// TIA Portal V19 export
FUNCTION_BLOCK "Area01_HU_FB"   // FB38, LAD
TITLE = AREA 01 HU PUMP
// stored: MemoryReserve 100, SetENOAutomatically false
   VAR_INPUT
      AreaInterface : "AreaInterface";
   END_VAR
   VAR_OUTPUT
      MachineInterface : "MachineInterface";
   END_VAR
   VAR
      Pump : "HU_Pump";
      Tank { S7_SetPoint := 'True'} : "HU_Tank";
      HMI : Struct
         Pressure_CoilCar : Real;
         Pressure_Peeler : Real;
         Pressure_JB_Cut : Real;
      END_STRUCT;
   END_VAR
   VAR_TEMP
      retval : Int;
      OilTemperature : Real;
      AnalTemperature_Real : Real;
      Delta : Real;
      Delta2 : Real;
   END_VAR
BEGIN

REGION Network 1: <<< PUMP >>>
END_REGION

REGION Network 2: Data In
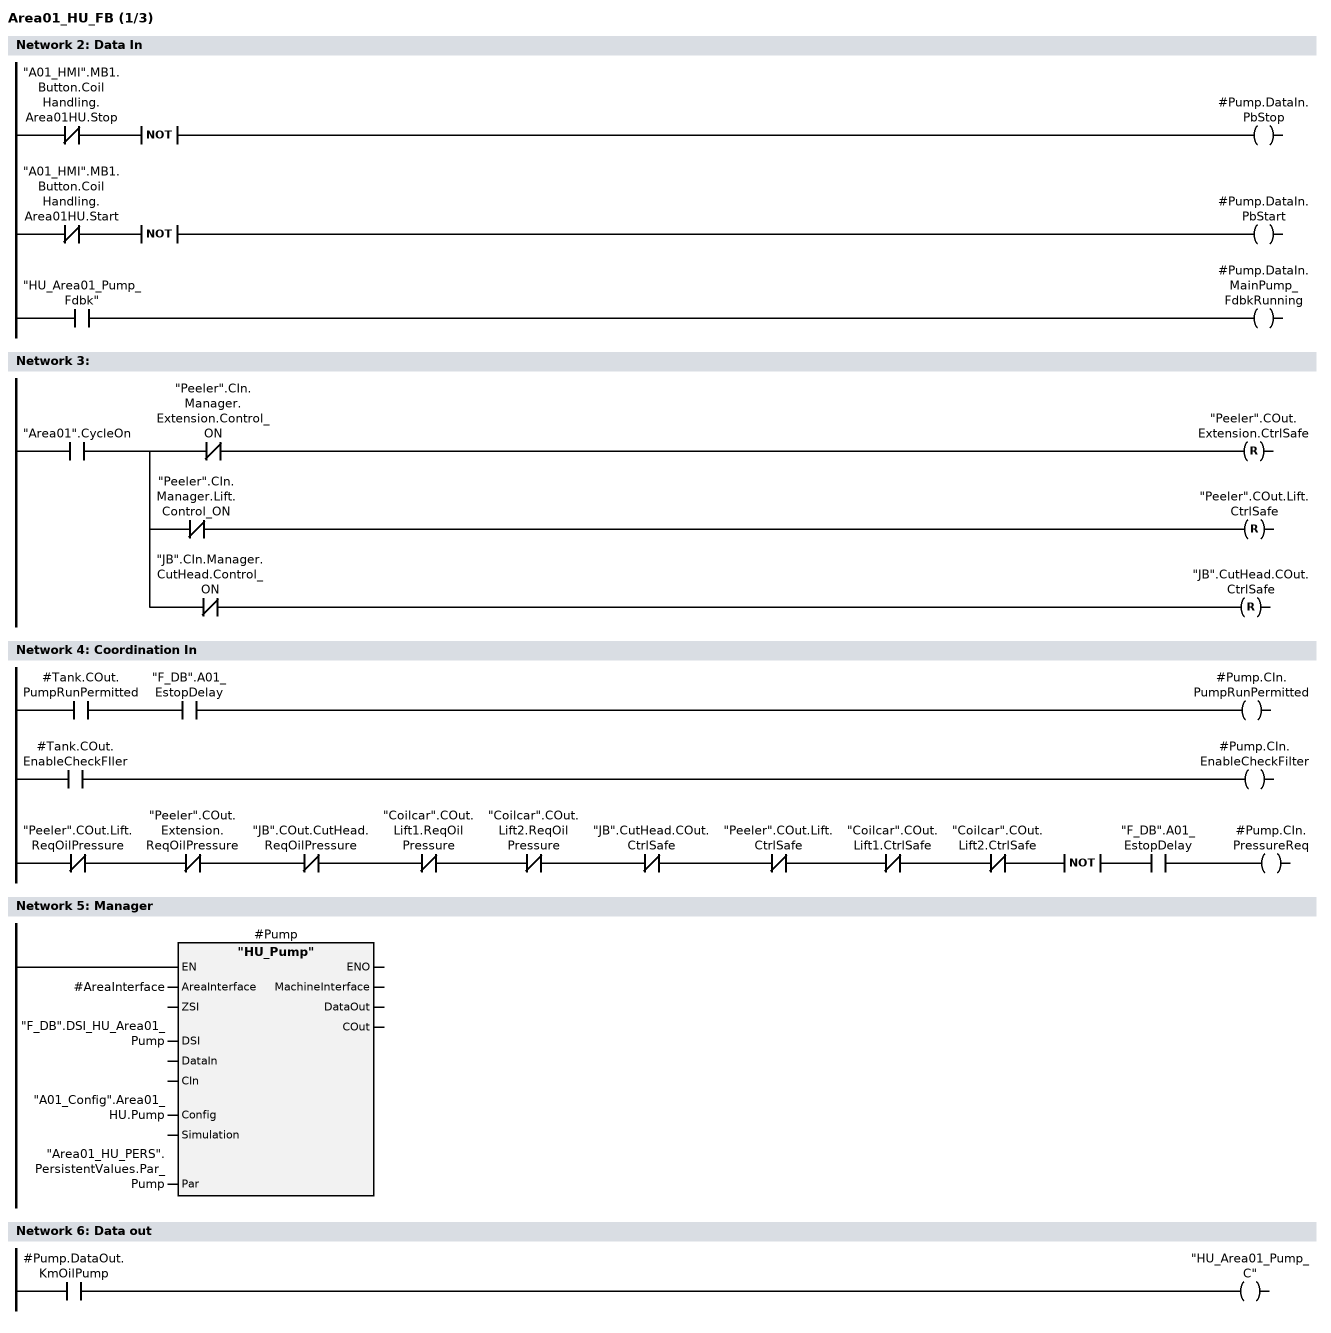
   RUNG wire#powerrail
      I_Contact( "A01_HMI".MB1.Button.CoilHandling.Area01HU.Stop )
      Not()
      Coil( #Pump.DataIn.PbStop )
   END_RUNG
   RUNG wire#powerrail
      I_Contact( "A01_HMI".MB1.Button.CoilHandling.Area01HU.Start )
      Not()
      Coil( #Pump.DataIn.PbStart )
   END_RUNG
   RUNG wire#powerrail
      Contact( "HU_Area01_Pump_Fdbk" )
      Coil( #Pump.DataIn.MainPump_FdbkRunning )
   END_RUNG
   // the same network as SCL:
   #Pump.DataIn.PbStop := NOT (NOT "A01_HMI".MB1.Button.CoilHandling.Area01HU.Stop);
   #Pump.DataIn.PbStart := NOT (NOT "A01_HMI".MB1.Button.CoilHandling.Area01HU.Start);
   #Pump.DataIn.MainPump_FdbkRunning := "HU_Area01_Pump_Fdbk";
END_REGION

REGION Network 3
   RUNG wire#powerrail
      Contact( "Area01".CycleOn )
      wire#w1
      I_Contact( "Peeler".CIn.Manager.Extension.Control_ON )
      R_Coil( "Peeler".COut.Extension.CtrlSafe )
   END_RUNG
   RUNG wire#w1
      I_Contact( "Peeler".CIn.Manager.Lift.Control_ON )
      R_Coil( "Peeler".COut.Lift.CtrlSafe )
   END_RUNG
   RUNG wire#w1
      I_Contact( "JB".CIn.Manager.CutHead.Control_ON )
      R_Coil( "JB".CutHead.COut.CtrlSafe )
   END_RUNG
   // the same network as SCL:
   IF "Area01".CycleOn AND NOT "Peeler".CIn.Manager.Extension.Control_ON THEN
       "Peeler".COut.Extension.CtrlSafe := FALSE;
   END_IF;
   IF "Area01".CycleOn AND NOT "Peeler".CIn.Manager.Lift.Control_ON THEN
       "Peeler".COut.Lift.CtrlSafe := FALSE;
   END_IF;
   IF "Area01".CycleOn AND NOT "JB".CIn.Manager.CutHead.Control_ON THEN
       "JB".CutHead.COut.CtrlSafe := FALSE;
   END_IF;
END_REGION

REGION Network 4: Coordination In
   RUNG wire#powerrail
      Contact( #Tank.COut.PumpRunPermitted )
      Contact( "F_DB".A01_EstopDelay )
      Coil( #Pump.CIn.PumpRunPermitted )
   END_RUNG
   RUNG wire#powerrail
      Contact( #Tank.COut.EnableCheckFIler )
      Coil( #Pump.CIn.EnableCheckFilter )
   END_RUNG
   RUNG wire#powerrail
      I_Contact( "Peeler".COut.Lift.ReqOilPressure )
      I_Contact( "Peeler".COut.Extension.ReqOilPressure )
      I_Contact( "JB".COut.CutHead.ReqOilPressure )
      I_Contact( "Coilcar".COut.Lift1.ReqOilPressure )
      I_Contact( "Coilcar".COut.Lift2.ReqOilPressure )
      I_Contact( "JB".CutHead.COut.CtrlSafe )
      I_Contact( "Peeler".COut.Lift.CtrlSafe )
      I_Contact( "Coilcar".COut.Lift1.CtrlSafe )
      I_Contact( "Coilcar".COut.Lift2.CtrlSafe )
      Not()
      Contact( "F_DB".A01_EstopDelay )
      Coil( #Pump.CIn.PressureReq )
   END_RUNG
   // the same network as SCL:
   #Pump.CIn.PumpRunPermitted := #Tank.COut.PumpRunPermitted AND "F_DB".A01_EstopDelay;
   #Pump.CIn.EnableCheckFilter := #Tank.COut.EnableCheckFIler;
   #Pump.CIn.PressureReq := NOT (NOT "Peeler".COut.Lift.ReqOilPressure AND NOT "Peeler".COut.Extension.ReqOilPressure AND NOT "JB".COut.CutHead.ReqOilPressure AND NOT "Coilcar".COut.Lift1.ReqOilPressure AND NOT "Coilcar".COut.Lift2.ReqOilPressure AND NOT "JB".CutHead.COut.CtrlSafe AND NOT "Peeler".COut.Lift.CtrlSafe AND NOT "Coilcar".COut.Lift1.CtrlSafe AND NOT "Coilcar".COut.Lift2.CtrlSafe) AND "F_DB".A01_EstopDelay;
END_REGION

REGION Network 5: Manager
   RUNG wire#powerrail
      #Pump(AreaInterface := #AreaInterface, ZSI :=, DSI := "F_DB".DSI_HU_Area01_Pump, DataIn :=, CIn :=, Config := "A01_Config".Area01_HU.Pump, Simulation :=, Par := "Area01_HU_PERS".PersistentValues.Par_Pump, MachineInterface =>, DataOut =>, COut =>)
   END_RUNG
   // the same network as SCL:
   #Pump(AreaInterface := #AreaInterface,   // "HU_Pump"
         DSI := "F_DB".DSI_HU_Area01_Pump,
         Config := "A01_Config".Area01_HU.Pump,
         Par := "Area01_HU_PERS".PersistentValues.Par_Pump);
END_REGION

REGION Network 6: Data out
   RUNG wire#powerrail
      Contact( #Pump.DataOut.KmOilPump )
      Coil( "HU_Area01_Pump_C" )
   END_RUNG
   // the same network as SCL:
   "HU_Area01_Pump_C" := #Pump.DataOut.KmOilPump;
END_REGION

REGION Network 7: >
END_REGION

REGION Network 8: >
END_REGION

REGION Network 9: >
END_REGION

REGION Network 10: <<< TANK >>>
END_REGION

REGION Network 11: Data In
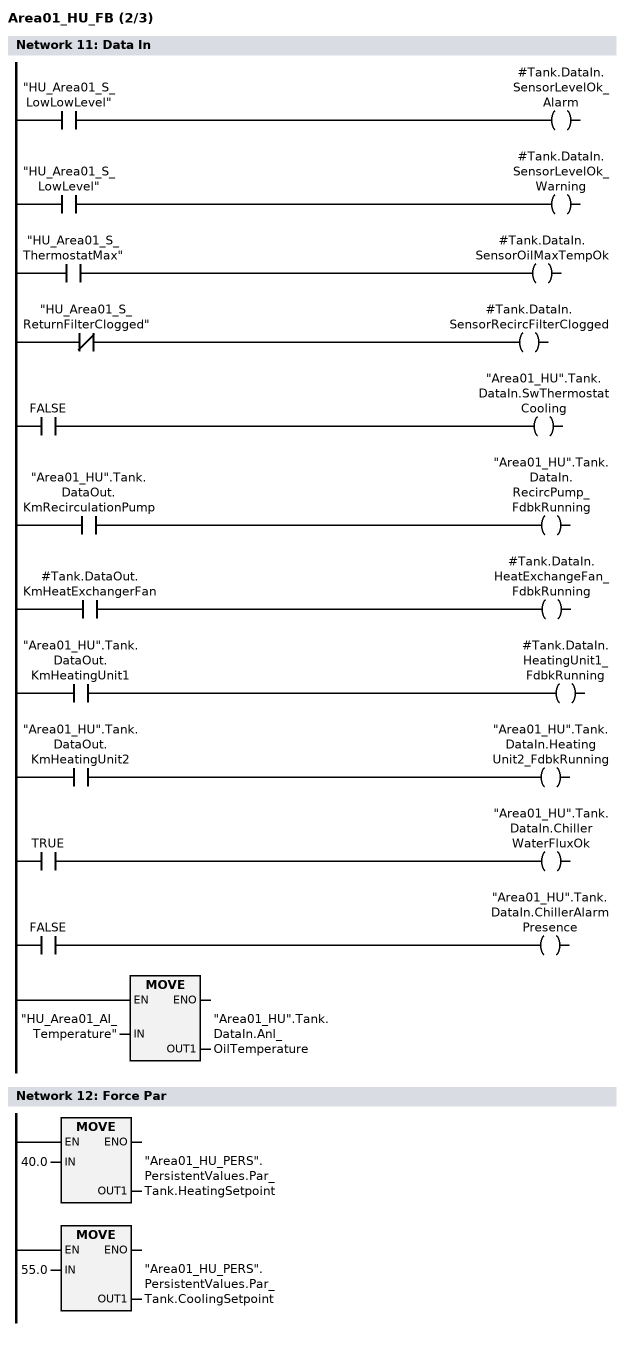
   RUNG wire#powerrail
      Contact( "HU_Area01_S_LowLowLevel" )
      Coil( #Tank.DataIn.SensorLevelOk_Alarm )
   END_RUNG
   RUNG wire#powerrail
      Contact( "HU_Area01_S_LowLevel" )
      Coil( #Tank.DataIn.SensorLevelOk_Warning )
   END_RUNG
   RUNG wire#powerrail
      Contact( "HU_Area01_S_ThermostatMax" )
      Coil( #Tank.DataIn.SensorOilMaxTempOk )
   END_RUNG
   RUNG wire#powerrail
      I_Contact( "HU_Area01_S_ReturnFilterClogged" )
      Coil( #Tank.DataIn.SensorRecircFilterClogged )
   END_RUNG
   RUNG wire#powerrail
      Contact( FALSE )
      Coil( "Area01_HU".Tank.DataIn.SwThermostatCooling )
   END_RUNG
   RUNG wire#powerrail
      Contact( "Area01_HU".Tank.DataOut.KmRecirculationPump )
      Coil( "Area01_HU".Tank.DataIn.RecircPump_FdbkRunning )
   END_RUNG
   RUNG wire#powerrail
      Contact( #Tank.DataOut.KmHeatExchangerFan )
      Coil( #Tank.DataIn.HeatExchangeFan_FdbkRunning )
   END_RUNG
   RUNG wire#powerrail
      Contact( "Area01_HU".Tank.DataOut.KmHeatingUnit1 )
      Coil( #Tank.DataIn.HeatingUnit1_FdbkRunning )
   END_RUNG
   RUNG wire#powerrail
      Contact( "Area01_HU".Tank.DataOut.KmHeatingUnit2 )
      Coil( "Area01_HU".Tank.DataIn.HeatingUnit2_FdbkRunning )
   END_RUNG
   RUNG wire#powerrail
      Contact( TRUE )
      Coil( "Area01_HU".Tank.DataIn.ChillerWaterFluxOk )
   END_RUNG
   RUNG wire#powerrail
      Contact( FALSE )
      Coil( "Area01_HU".Tank.DataIn.ChillerAlarmPresence )
   END_RUNG
   RUNG wire#powerrail
      Move(in := "HU_Area01_AI_Temperature", out1 => "Area01_HU".Tank.DataIn.Anl_OilTemperature)
   END_RUNG
   // the same network as SCL:
   #Tank.DataIn.SensorLevelOk_Alarm := "HU_Area01_S_LowLowLevel";
   #Tank.DataIn.SensorLevelOk_Warning := "HU_Area01_S_LowLevel";
   #Tank.DataIn.SensorOilMaxTempOk := "HU_Area01_S_ThermostatMax";
   #Tank.DataIn.SensorRecircFilterClogged := NOT "HU_Area01_S_ReturnFilterClogged";
   "Area01_HU".Tank.DataIn.SwThermostatCooling := FALSE;
   "Area01_HU".Tank.DataIn.RecircPump_FdbkRunning := "Area01_HU".Tank.DataOut.KmRecirculationPump;
   #Tank.DataIn.HeatExchangeFan_FdbkRunning := #Tank.DataOut.KmHeatExchangerFan;
   #Tank.DataIn.HeatingUnit1_FdbkRunning := "Area01_HU".Tank.DataOut.KmHeatingUnit1;
   "Area01_HU".Tank.DataIn.HeatingUnit2_FdbkRunning := "Area01_HU".Tank.DataOut.KmHeatingUnit2;
   "Area01_HU".Tank.DataIn.ChillerWaterFluxOk := TRUE;
   "Area01_HU".Tank.DataIn.ChillerAlarmPresence := FALSE;
   "Area01_HU".Tank.DataIn.Anl_OilTemperature := "HU_Area01_AI_Temperature";
END_REGION

REGION Network 12: Force Par
   RUNG wire#powerrail
      { S7_GenerateENO := "TRUE" } Move(in := 40.0, out1 => "Area01_HU_PERS".PersistentValues.Par_Tank.HeatingSetpoint)
   END_RUNG
   RUNG wire#powerrail
      { S7_GenerateENO := "TRUE" } Move(in := 55.0, out1 => "Area01_HU_PERS".PersistentValues.Par_Tank.CoolingSetpoint)
   END_RUNG
   // the same network as SCL:
   "Area01_HU_PERS".PersistentValues.Par_Tank.HeatingSetpoint := 40.0;
   "Area01_HU_PERS".PersistentValues.Par_Tank.CoolingSetpoint := 55.0;
END_REGION

REGION Network 13: HMI pressure
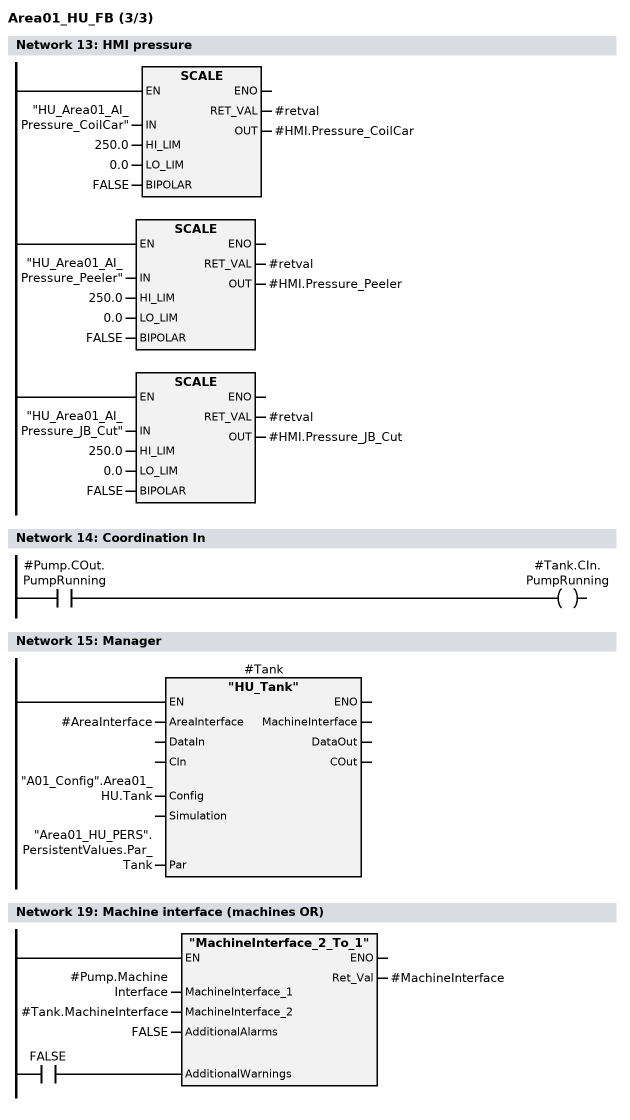
   #retval := SCALE(IN := "HU_Area01_AI_Pressure_CoilCar",
                    HI_LIM := 250.0,
                    LO_LIM := 0.0,
                    BIPOLAR := FALSE,
                    OUT => #HMI.Pressure_CoilCar);
   #retval := SCALE(IN := "HU_Area01_AI_Pressure_Peeler",
                    HI_LIM := 250.0,
                    LO_LIM := 0.0,
                    BIPOLAR := FALSE,
                    OUT => #HMI.Pressure_Peeler);
   #retval := SCALE(IN := "HU_Area01_AI_Pressure_JB_Cut",
                    HI_LIM := 250.0,
                    LO_LIM := 0.0,
                    BIPOLAR := FALSE,
                    OUT => #HMI.Pressure_JB_Cut);
END_REGION

REGION Network 14: Coordination In
   RUNG wire#powerrail
      Contact( #Pump.COut.PumpRunning )
      Coil( #Tank.CIn.PumpRunning )
   END_RUNG
   // the same network as SCL:
   #Tank.CIn.PumpRunning := #Pump.COut.PumpRunning;
END_REGION

REGION Network 15: Manager
   RUNG wire#powerrail
      #Tank(AreaInterface := #AreaInterface, DataIn :=, CIn :=, Config := "A01_Config".Area01_HU.Tank, Simulation :=, Par := "Area01_HU_PERS".PersistentValues.Par_Tank, MachineInterface =>, DataOut =>, COut =>)
   END_RUNG
   // the same network as SCL:
   #Tank(AreaInterface := #AreaInterface,   // "HU_Tank"
         Config := "A01_Config".Area01_HU.Tank,
         Par := "Area01_HU_PERS".PersistentValues.Par_Tank);
END_REGION

REGION Network 16: >
END_REGION

REGION Network 17: >
END_REGION

REGION Network 18: >
END_REGION

REGION Network 19: Machine interface (machines OR)
   RUNG wire#powerrail
      "MachineInterface_2_To_1"(AdditionalWarnings := wire#w1, MachineInterface_1 := #Pump.MachineInterface, MachineInterface_2 := #Tank.MachineInterface, AdditionalAlarms := FALSE, Ret_Val => #MachineInterface)
   END_RUNG
   RUNG wire#powerrail
      Contact( FALSE )
   END_RUNG wire#w1
   // the same network as SCL:
   #MachineInterface := "MachineInterface_2_To_1"(MachineInterface_1 := #Pump.MachineInterface,
                           MachineInterface_2 := #Tank.MachineInterface,
                           AdditionalAlarms := FALSE,
                           AdditionalWarnings := FALSE);
END_REGION
END_FUNCTION_BLOCK
